// TwinCAT 3 PLC project Motoransteuerung
// ProgramVersion: 3.1.4022.0
// libraries:
//   Tc2_MC2, * (Beckhoff Automation GmbH)
//   Tc2_Standard, * (Beckhoff Automation GmbH)
//   Tc2_System, * (Beckhoff Automation GmbH)
//   Tc3_Module, * (Beckhoff Automation GmbH)
// project tree:
//   DUTs/ EnumState.TcDUT
//   / PlcTask.TcTTO
//   POUs/ MAIN.TcPOU
// (motion and I/O tree: see PLC project shutdown)
// real-time tasks:
//   TASK Plc_Task: cycle T#10ms, priority 20, ADS port 350
//   TASK IrSensor_Task: cycle T#5ms, priority 9, ADS port 351
//   TASK UDP_Task: cycle T#10ms, priority 10, ADS port 354
// variable links:
//   Motoransteuerung/Motoransteuerung Instance <-> Antriebe und Greifer/Axes/Achse 1
//     PlcTask Inputs/MAIN.axis1.NcToPlc <-> Outputs/ToPlc
//     PlcTask Outputs/MAIN.axis1.PlcToNc <-> Inputs/FromPlc
//   Motoransteuerung/Motoransteuerung Instance <-> Antriebe und Greifer/Axes/Achse 2
//     PlcTask Inputs/MAIN.axis2.NcToPlc <-> Outputs/ToPlc
//     PlcTask Outputs/MAIN.axis2.PlcToNc <-> Inputs/FromPlc
//   Motoransteuerung/Motoransteuerung Instance <-> Antriebe und Greifer/Axes/Achse 3
//     PlcTask Inputs/MAIN.axis3.NcToPlc <-> Outputs/ToPlc
//     PlcTask Outputs/MAIN.axis3.PlcToNc <-> Inputs/FromPlc

CONFIGURATION Motoransteuerung
    RESOURCE PLC ON TwinCAT3
        TASK PlcTask(INTERVAL := T#5ms, PRIORITY := 2);
        PROGRAM MAIN WITH PlcTask : MAIN;
    END_RESOURCE
END_CONFIGURATION

// ---- DUTs/EnumState.TcDUT
{attribute 'qualified_only'}
{attribute 'strict'}
TYPE EnumState :
(
	init,
	drive1,
	drive2,
	reset
);
END_TYPE

// ---- POUs/MAIN.TcPOU
PROGRAM MAIN
VAR
	//Achsen Referenzen
	axis1: AXIS_REF;
	axis2: AXIS_REF;
	axis3: AXIS_REF;
	
	//Objekte um Achsen anzusteuern
	powerAxis1: MC_Power;
	driveAxis11: MC_MoveVelocity;
	driveAxis12: MC_MoveVelocity;
	resetAxis1: MC_Reset;
	
	powerAxis2: MC_Power;
	driveAxis21: MC_MoveVelocity;
	driveAxis22: MC_MoveVelocity;
	resetAxis2: MC_Reset;
	
	powerAxis3: MC_Power;
	driveAxis31: MC_MoveVelocity;
	driveAxis32: MC_MoveVelocity;
	resetAxis3: MC_Reset;
	
	//Achse Freischalten, Regler Freischalten
	enableControl: BOOL	:=0;
	enablePos: BOOL		:=0;
	enableNeg: BOOL		:=0;
	override:  LREAL	:=0;
	
	//Fahrbefehl Ausführen
	drive1Execute: BOOL	:=0;
	drive2Execute: BOOL	:=0;
	
	//State Maschine
	nextState:EnumState	:=EnumState.init;
	state:EnumState		:=EnumState.init;
	
	//Stellgeschwindigkeit und Richtung
	velocity1:	LREAL	:=0;
	velocity2:	LREAL	:=0;
	velocity3:	LREAL	:=0;
	
	direction1:	MC_Direction:=MC_Positive_Direction;
	direction2:	MC_Direction:=MC_Positive_Direction;
	direction3:	MC_Direction:=MC_Positive_Direction;
	
	delay:TON;
	
END_VAR

axis1.ReadStatus();
axis2.ReadStatus();
axis3.ReadStatus();

//Zu Ersetzen mit SwitchCase
//powerAxis1(Axis:=axis1,Enable:=enableControl,Enable_Positive:=enablePos,Enable_Negative:=enableNeg,Override:=override);
//IF powerAxis1.Status THEN
//	moveAxis1(Axis:=axis1,Velocity:=250,Direction:=MC_Positive_Direction,Execute:=1,BufferMode:=MC_Buffered);
//END_IF
//Zu Ersetzen mit SwitchCase

CASE state OF
	EnumState.init:
		enableControl:=1;
		enablePos:=1;
		enableNeg:=1;
		override:=100;
		
		powerAxis1(Axis:=axis1,Enable:=enableControl,Enable_Positive:=enablePos,Enable_Negative:=enableNeg,Override:=override);
		powerAxis2(Axis:=axis2,Enable:=enableControl,Enable_Positive:=enablePos,Enable_Negative:=enableNeg,Override:=override);
		powerAxis3(Axis:=axis3,Enable:=enableControl,Enable_Positive:=enablePos,Enable_Negative:=enableNeg,Override:=override);
		
		IF (powerAxis1.Status AND powerAxis2.Status AND powerAxis3.Status) THEN	
			nextState:=EnumState.drive1; 
			drive1Execute:=1;
		END_IF
		IF (powerAxis1.Error OR powerAxis2.Error OR powerAxis3.Error) THEN
			nextState:=EnumState.reset;
		END_IF
		
	EnumState.drive1:
	
		driveAxis11(Axis:=axis1,Velocity:=250,Direction:=direction1,Execute:=drive1Execute,BufferMode:=MC_Buffered);
		driveAxis21(Axis:=axis2,Velocity:=250,Direction:=direction2,Execute:=drive1Execute,BufferMode:=MC_Buffered);
		driveAxis31(Axis:=axis3,Velocity:=250,Direction:=direction3,Execute:=drive1Execute,BufferMode:=MC_Buffered);
		
		
		IF (powerAxis1.Error OR powerAxis2.Error OR powerAxis3.Error) THEN
			nextState:=EnumState.reset;
		END_IF
		
	EnumState.drive2:
	
		driveAxis11(Axis:=axis1,Velocity:=900,Direction:=direction1,Execute:=drive2Execute,BufferMode:=MC_Buffered);
		driveAxis21(Axis:=axis2,Velocity:=900,Direction:=direction2,Execute:=drive2Execute,BufferMode:=MC_Buffered);
		driveAxis31(Axis:=axis3,Velocity:=900,Direction:=direction3,Execute:=drive2Execute,BufferMode:=MC_Buffered);
		
		IF (powerAxis1.Error OR powerAxis2.Error OR powerAxis3.Error) THEN
			nextState:=EnumState.reset;
		END_IF	
	EnumState.reset:;
	ELSE
		nextState:=EnumState.reset;
END_CASE
state:=nextState;

END_PROGRAM
